TYPE DUT_NC_Kanal :
STRUCT
	AxTo3DOK			:BOOL;
	AxToPTPOK			:BOOL;

	Ready				:BOOL;
	Aktiv				:BOOL;
	Run					:BOOL;
	Err					:BOOL;

	MFuncNr				:INT;
	MFuncReq			:BOOL;
	MFuncQuittNr		:INT;
	MFuncQuitt			:BOOL;

END_STRUCT
END_TYPE

(* stored: Version 1.1.0.1
   DUT DUT_NC_Kanal: Id {f3f2cf34-b99a-4ec6-94c0-473a6b00c70c} *)
